FUNCTION_BLOCK SkillRotatingArmController (* Basic Function Block Type *)
  (* Standard: 61499-2 *)
  (* Version 0.0, 2/16/2024, midxav, Template *)
  PACKAGE Main;
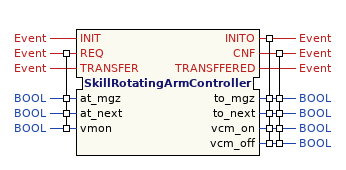
  EVENT_INPUT
    INIT; (* Initialization Request *)
    REQ WITH at_mgz, at_next, vmon; (* Normal Execution Request *)
    TRANSFER;
  END_EVENT
  EVENT_OUTPUT
    INITO WITH to_mgz, to_next, vcm_on, vcm_off; (* Initialization Confirm *)
    CNF WITH to_mgz, to_next, vcm_on, vcm_off; (* Execution Confirmation *)
    TRANSFFERED;
  END_EVENT
  VAR_INPUT
    at_mgz : BOOL;
    at_next : BOOL;
    vmon : BOOL;
  END_VAR
  VAR_OUTPUT
    to_mgz : BOOL;
    to_next : BOOL;
    vcm_on : BOOL;
    vcm_off : BOOL;
  END_VAR
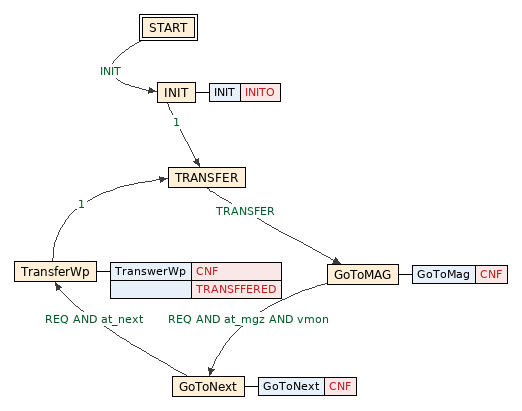
  EC_STATES
    START; (* Initial State *)
    INIT : INIT -> INITO; (* Initialization *)
    GoToMAG : GoToMag -> CNF;
    GoToNext : GoToNext -> CNF;
    TransferWp : TranswerWp -> CNF, -> TRANSFFERED;
    TRANSFER;
  END_STATES
  EC_TRANSITIONS
    START TO INIT := INIT;
    TRANSFER TO GoToMAG := TRANSFER;
    GoToMAG TO GoToNext := REQ AND at_mgz AND vmon;
    GoToNext TO TransferWp := REQ AND at_next;
    TransferWp TO TRANSFER := 1;
    INIT TO TRANSFER := 1;
  END_TRANSITIONS
  ALGORITHM INIT IN ST: (* Initialization algorithm *)
to_mgz :=FALSE;
to_next :=TRUE;
vcm_on := FALSE;
vcm_off := TRUE;
  END_ALGORITHM
  ALGORITHM GoToMag IN ST:
to_mgz := TRUE;
to_next := FALSE;
vcm_on := TRUE;
vcm_off := FALSE;
  END_ALGORITHM
  ALGORITHM GoToNext IN ST:
to_mgz := FALSE;
to_next := TRUE;
  END_ALGORITHM
  ALGORITHM TranswerWp IN ST:
vcm_on := FALSE;
vcm_off := TRUE;
  END_ALGORITHM
END_FUNCTION_BLOCK
